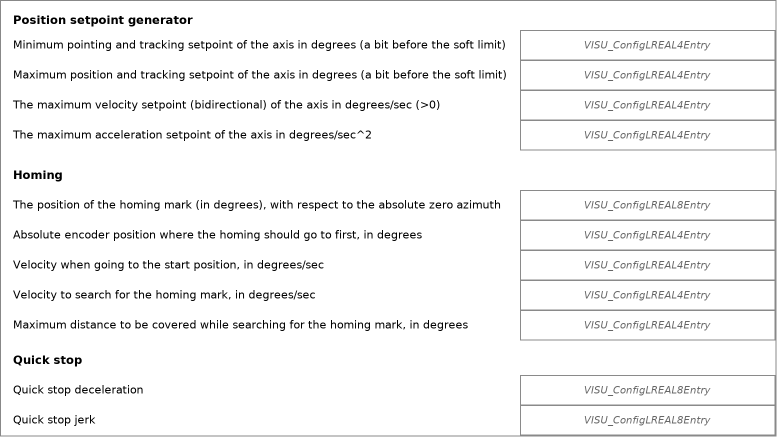
VISUALIZATION VISU_AxesConfig_Azimuth_2  // 777x437
VAR_IN_OUT
    active : AxesAzimuthConfig;
    editable : AxesAzimuthConfig;
END_VAR
    Frame (520,190 255x30)
        shows VISU_ConfigLREAL8Entry(active := active.homingHomePosition, editable := editable.homingHomePosition)
    Label (10,5 205x30), "Position setpoint generator"
    Label (10,30 500x30), "Minimum pointing and tracking setpoint of the axis in degrees (a bit before the soft limit)"
    Frame (520,30 255x30)
        shows VISU_ConfigLREAL4Entry(active := active.minPositionSetpoint, editable := editable.minPositionSetpoint)
    Label (10,60 500x30), "Maximum position and tracking setpoint of the axis in degrees (a bit before the soft limit)"
    Label (10,90 475x30), "The maximum velocity setpoint (bidirectional) of the axis in degrees/sec (>0)"
    Label (10,120 475x30), "The maximum acceleration setpoint of the axis in degrees/sec^2"
    Label (10,160 205x30), "Homing"
    Label (10,220 475x30), "Absolute encoder position where the homing should go to first, in degrees"
    Label (10,250 475x30), "Velocity when going to the start position, in degrees/sec"
    Label (10,280 505x30), "Velocity to search for the homing mark, in degrees/sec"
    Label (10,310 500x30), "Maximum distance to be covered while searching for the homing mark, in degrees"
    Frame (520,60 255x30)
        shows VISU_ConfigLREAL4Entry(active := active.maxPositionSetpoint, editable := editable.maxPositionSetpoint)
    Frame (520,90 255x30)
        shows VISU_ConfigLREAL4Entry(active := active.maxVelocitySetpoint, editable := editable.maxVelocitySetpoint)
    Frame (520,120 255x30)
        shows VISU_ConfigLREAL4Entry(active := active.maxAccelerationSetpoint, editable := editable.maxAccelerationSetpoint)
    Frame (520,220 255x30)
        shows VISU_ConfigLREAL4Entry(active := active.homingStartAbsEncPosition, editable := editable.homingStartAbsEncPosition)
    Frame (520,250 255x30)
        shows VISU_ConfigLREAL4Entry(active := active.homingGotoStartVelocity, editable := editable.homingGotoStartVelocity)
    Frame (520,280 255x30)
        shows VISU_ConfigLREAL4Entry(active := active.homingVelocity, editable := editable.homingVelocity)
    Frame (520,310 255x30)
        shows VISU_ConfigLREAL4Entry(active := active.homingRange, editable := editable.homingRange)
    Label (10,190 500x30), "The position of the homing mark (in degrees), with respect to the absolute zero azimuth"
    Label (10,345 205x30), "Quick stop"
    Frame (520,375 255x30)
        shows VISU_ConfigLREAL8Entry(active := active.quickStopDeceleration, editable := editable.quickStopDeceleration)
    Label (10,375 500x30), "Quick stop deceleration"
    Label (10,405 500x30), "Quick stop jerk"
    Frame (520,405 255x30)
        shows VISU_ConfigLREAL8Entry(active := active.quickStopJerk, editable := editable.quickStopJerk)
END_VISUALIZATION

(* stored: Version 1.1.0.1, ProductVersion 3.1.4019.2
   Visu VISU_AxesConfig_Azimuth_2: Id {7c433477-a215-4448-ac79-621430c43b1a} *)
